(* PLC project Unnamed, Unknown Unnamed 1 *)
(* stored: creationDateTime 2026-02-02T21:22:35, modificationDateTime 2026-02-02T21:22:35 *)

PROGRAM main
  VAR
    IN_ON AT %IX0.3 : BOOL;
    OUT AT %QX0.0 : BOOL;
    IN_OFF AT %IX0.4 : BOOL;
  END_VAR
  VAR
    LocalVar : DINT;
  END_VAR
  VAR  (* added by the conversion: wires and edge detectors of the diagram *)
    R_TRIG1 : R_TRIG;
  END_VAR

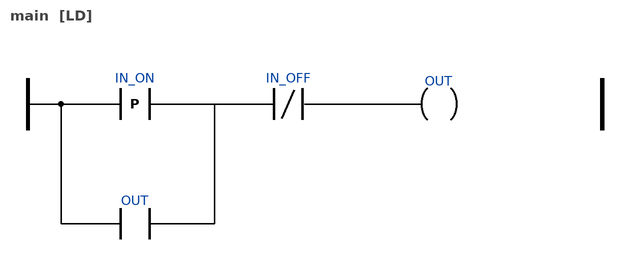
(* LD diagram, written out as Structured Text *)
R_TRIG1(CLK := IN_ON);
OUT := (R_TRIG1.Q OR OUT) AND NOT IN_OFF;
END_PROGRAM

CONFIGURATION Config0
  RESOURCE Res0 ON PLC
    TASK task0(INTERVAL := T#20ms, PRIORITY := 1);
    PROGRAM instance0 WITH task0 : main;
  END_RESOURCE
END_CONFIGURATION
